FUNCTION_BLOCK Sensor_StateOrder_subView
  (* Version 0.1, 2005-12-14, Oscar Ljungkrantz, Chalmers *)
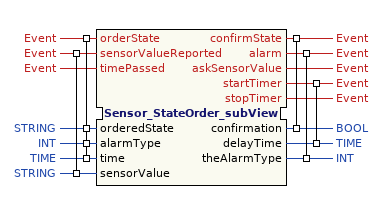
  EVENT_INPUT
    orderState WITH orderedState, alarmType, time;
    sensorValueReported WITH sensorValue;
    timePassed;
  END_EVENT
  EVENT_OUTPUT
    confirmState WITH confirmation;
    alarm WITH theAlarmType;
    askSensorValue;
    startTimer WITH delayTime;
    stopTimer;
  END_EVENT
  VAR_INPUT
    orderedState : STRING;
    alarmType : INT;
    time : TIME;
    sensorValue : STRING;
  END_VAR
  VAR_OUTPUT
    confirmation : BOOL;
    delayTime : TIME;
    theAlarmType : INT;
  END_VAR
  VAR
    currentOrderedState : STRING;
    currentAlarmType : INT := 1;
    operating : BOOL := FALSE;
  END_VAR
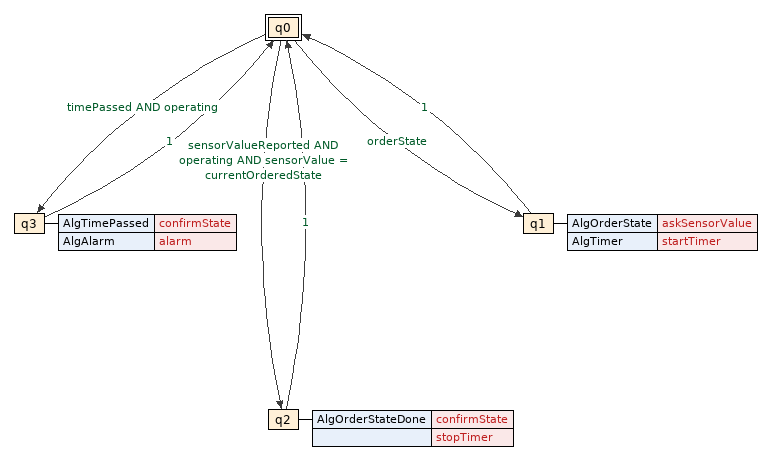
  EC_STATES
    q0;
    q1 : AlgOrderState -> askSensorValue, AlgTimer -> startTimer;
    q2 : AlgOrderStateDone -> confirmState, -> stopTimer;
    q3 : AlgTimePassed -> confirmState, AlgAlarm -> alarm;
  END_STATES
  EC_TRANSITIONS
    q0 TO q1 := orderState;
    q1 TO q0 := 1;
    q0 TO q2 := sensorValueReported AND operating AND sensorValue = currentOrderedState;
    q2 TO q0 := 1;
    q0 TO q3 := timePassed AND operating;
    q3 TO q0 := 1;
  END_TRANSITIONS
  ALGORITHM AlgOrderState IN Java:
		currentOrderedState = orderedState;
		currentAlarmType = alarmType;
		operating = TRUE;
  END_ALGORITHM
  ALGORITHM AlgTimer IN Java:
		delayTime = time;
  END_ALGORITHM
  ALGORITHM AlgOrderStateDone IN Java:
		confirmation = TRUE;
		operating = FALSE;
  END_ALGORITHM
  ALGORITHM AlgTimePassed IN Java:
		confirmation = FALSE;
  END_ALGORITHM
  ALGORITHM AlgAlarm IN Java:
		theAlarmType = currentAlarmType;
  END_ALGORITHM
END_FUNCTION_BLOCK
(* other elements stored in the file *)
(* In a sensor the time is an input instead of a property (local variable) as in the actuator *)
(* __Not needed for a sensor__ Event Name="orderActuator"> <With Var="actuatorValue" /> </Event *)
(* __Not needed for a sensor__ Event Name="setOperationStatus"> <With Var="isIdle" /> </Event *)
(* __Not needed for a sensor__ VarDeclaration Name="actuatorValue" Type="STRING" / *)
(* __Not needed for a sensor__ VarDeclaration Name="isIdle" Type="BOOL" / *)
(* In a sensor you can ask the value of the sensor directly *)
(* __Not needed for a sensor__ ECAction Algorithm="AlgIsOperating" Output="setOperationStatus" / *)
(* __Not needed (since it is stated above) for a sensor__ ECAction Output="askSensorValue" / *)
(* __Not needed for a sensor__ ECAction Algorithm="AlgIsNotOperating" Output="setOperationStatus" / *)
(* __Not needed for a sensor__ Algorithm Name="IsOperating"> <Other Language="Java" Text= " isIdle = FALSE; operating = TRUE; " /> </Algorithm *)
(* __Not needed for a sensor__ Algorithm Name="AlgIsNotOperating"> <Other Language="Java" Text= " isIdle = TRUE; operating = FALSE; " /> </Algorithm *)
